(* Logix 5000 project; controller ProyectoIntegrador Emulate 5570 rev 30.11; software revision 30.00 *)

TASK MainTask (continuous, watchdog 500 ms) : MainProgram

MODULES
   Local : Emulate 5570 (ICP 2, rev 30.11)
      IO_module : vendor 1 type 0 code 15 (ICP 3, rev 1.1, Output RPI 150 ms)
END_MODULES

PROGRAM MainProgram   (* main routine MainRoutine *)
VAR
   Action_000 : SFC_ACTION := (Status := 16#0020_0000, PauseTimer := 1);
   Action_001 : SFC_ACTION := (Status := 16#0020_0000, PauseTimer := 1);
   Action_002 : SFC_ACTION := (Status := 16#0020_0000, PauseTimer := 1);
   Action_003 : SFC_ACTION := (Status := 16#0020_0000, PauseTimer := 1);
   Action_004 : SFC_ACTION := (Status := 16#0020_0000, PauseTimer := 1);
   Action_005 : SFC_ACTION := (Status := 16#0020_0000, PauseTimer := 1);
   Action_006 : SFC_ACTION := (Status := 16#0020_0000, PauseTimer := 1);
   Action_007 : SFC_ACTION := (Status := 16#0020_0000, PauseTimer := 1);
   Action_008 : SFC_ACTION := (Status := 16#0020_0000, PauseTimer := 1);
   Action_009 : SFC_ACTION := (Status := 16#0020_0000, PauseTimer := 1);
   Action_010 : SFC_ACTION := (Status := 16#0020_0000, PauseTimer := 1);
   Action_011 : SFC_ACTION := (Status := 16#0020_0000, PauseTimer := 1);
   Action_012 : SFC_ACTION := (Status := 16#0020_0000, PauseTimer := 1);
   Action_013 : SFC_ACTION := (Status := 16#0020_0000, PauseTimer := 1);
   Action_014 : SFC_ACTION := (Status := 16#0020_0000, PauseTimer := 1);
   C1b : BOOL;   // Moves Cilinder 1 backward
   C1f : BOOL;   // Move cilinder 1 forward
   C2b : DINT;   // Move the cilinder 2 backwards
   C2f : BOOL;   // Move the cilinder 2 forward
   Clasif : BOOL;   // Encender/Apagar Classificador
   Compressor : BOOL;   // Encender/Apagar Compressor
   Lavdo : BOOL;   // Encender/Apagar Lavado
   lConv : BOOL;   // Sensor de cajas conveyor belt 3 (vegetal grande)
   lCount : DINT;   // Large box counter
   mConv : BOOL;
   mCount : DINT;   // Medium Boxes count
   RC5 : BOOL;   // Encender/Apagar roller conveyor 4
   RC_1 : BOOL;   // Encender/Apagar roller conveyor 1
   RC_2 : BOOL;   // Encender/Apagar roller conveyor 2
   RC_3 : BOOL;   // Encender/Apagar roller conveyor 3
   RC_4 : BOOL;   // Encender/Apagar roller conveyor 4
   S1_C1 : BOOL;   // Cilindro 1 recogido
   S1_C2 : BOOL;   // Sensor 1 final de carrera cilindro2
   S2_C1 : BOOL;   // Sensor 2 final de carrera cilindro 1
   S2_C2 : BOOL;   // Sensor 2 final de carrera cilindro 2
   S_clasif : DINT;   // Sensor para clasificacion de empaque
   sConv : BOOL;
   sCount : DINT;   // Small Boxes Count
   Secado : BOOL;   // Encender/Apagar Secado
   Start : BOOL;   // Inicio del proceso
   Step_000 : SFC_STEP := (Status := 16#0020_0000, PauseTimer := 1);
   Step_001 : SFC_STEP := (Status := 16#0020_0000, PauseTimer := 1);
   Step_002 : SFC_STEP := (Status := 16#0020_0000, PauseTimer := 1);
   Step_003 : SFC_STEP := (Status := 16#0020_0000, PauseTimer := 1);
   Step_004 : SFC_STEP := (Status := 16#0020_0000, PauseTimer := 1);
   Step_005 : SFC_STEP := (Status := 16#0020_0000, PauseTimer := 1);
   Step_006 : SFC_STEP := (Status := 16#0020_0000, PauseTimer := 1);
   Step_007 : SFC_STEP := (Status := 16#0020_0000, PauseTimer := 1);
   Step_008 : SFC_STEP := (Status := 16#0020_0000, PauseTimer := 1);
   Step_009 : SFC_STEP := (Status := 16#0020_0000, PauseTimer := 1);
   Step_010 : SFC_STEP := (Status := 16#0020_0000, PauseTimer := 1);
   Step_011 : SFC_STEP := (Status := 16#0020_0000, PauseTimer := 1);
   Step_012 : SFC_STEP := (Status := 16#0020_0000, PauseTimer := 1);
   Step_013 : SFC_STEP := (Status := 16#0020_0000, PauseTimer := 1);
   Step_014 : SFC_STEP := (Status := 16#0020_0000, PauseTimer := 1);
   Step_015 : SFC_STEP := (Status := 16#0020_0000, PauseTimer := 1);
   Step_016 : SFC_STEP := (Status := 16#0020_0000, PauseTimer := 1);
   Step_017 : SFC_STEP := (Status := 16#0020_0000, PauseTimer := 1);
   Step_018 : SFC_STEP := (Status := 16#0020_0000, PauseTimer := 1);
   Step_021 : SFC_STEP := (Status := 16#0020_0000, PauseTimer := 1);
   Step_022 : SFC_STEP := (Status := 16#0020_0000, PauseTimer := 1);
   Step_023 : SFC_STEP := (Status := 16#0020_0000, PauseTimer := 1);
   Step_024 : SFC_STEP := (Status := 16#0020_0000, PauseTimer := 1);
   Step_025 : SFC_STEP := (Status := 16#0020_0000, PauseTimer := 1);
   Step_031 : SFC_STEP := (Status := 16#0020_0000, PauseTimer := 1);
   Step_041 : SFC_STEP := (Status := 16#0020_0000, PauseTimer := 1);
   Step_042 : SFC_STEP := (Status := 16#0020_0000, PauseTimer := 1);
   Step_100 : SFC_STEP := (Status := 16#0020_0000, PauseTimer := 1);
   Step_101 : SFC_STEP := (Status := 16#0020_0000, PauseTimer := 1);
   Step_102 : SFC_STEP := (Status := 16#0020_0000, PauseTimer := 1);
   Step_103 : SFC_STEP := (Status := 16#0020_0000, PauseTimer := 1);
   Stop : BOOL;   // Stop Button
   Tran_000 : BOOL;
   Tran_001 : BOOL;
   Tran_002 : BOOL;
   Tran_003 : BOOL;
   Tran_004 : BOOL;
   Tran_005 : BOOL;
   Tran_006 : BOOL;
   Tran_007 : BOOL;
   Tran_008 : BOOL;
   Tran_009 : BOOL;
   Tran_010 : BOOL;
   Tran_011 : BOOL;
   Tran_012 : BOOL;
   Tran_016 : BOOL;
   Tran_017 : BOOL;
   Tran_018 : BOOL;
   Tran_019 : BOOL;
   Volcar : BOOL;   // Encendr/Apagar volcador
END_VAR

ROUTINE Distribution   (* sequential function chart *)
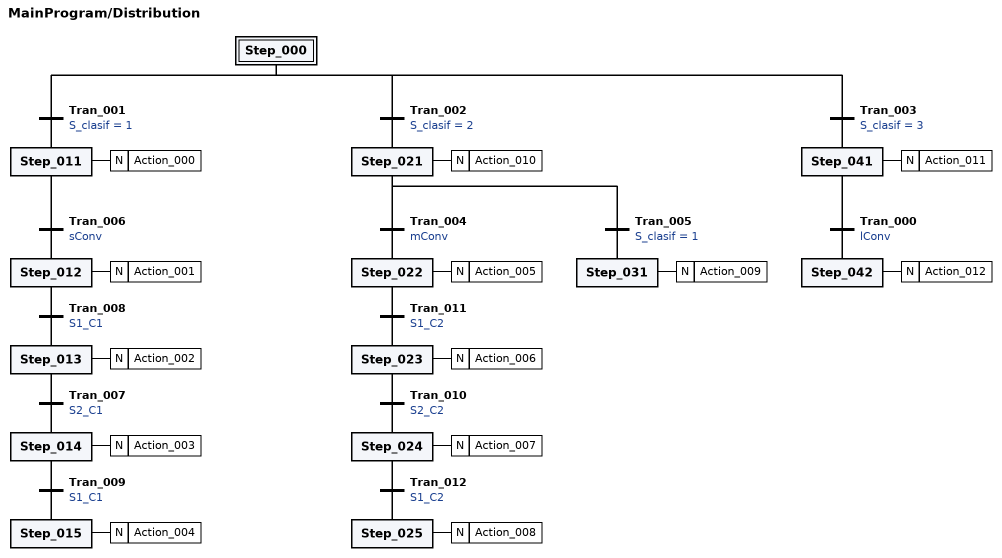
   // If the boxes
   // are medium
   // If the boxes
   // are small
   // If the boxes
   // are large
   // Sink
   // Transition
   // Pneumatic
   // divider G7
   // Sink
   // Transition
   // Sink
   // Transition
   // Discuss
   // with group
   // !!!
   // Should we have BC1, BC2 and BC3 always
   // turned on ??
   INITIAL_STEP Step_000:
   END_STEP
   TRANSITION Tran_001 FROM Step_000 TO Step_011
      := S_clasif = 1
         
   END_TRANSITION
   TRANSITION Tran_002 FROM Step_000 TO Step_021
      := S_clasif = 2
         
   END_TRANSITION
   TRANSITION Tran_003 FROM Step_000 TO Step_041
      := S_clasif = 3
         
   END_TRANSITION
   STEP Step_011:
      ACTION Action_000 (N):
         (* Move the rolling
         conveyor 5 forward*)
         RC5 := 1;
      END_ACTION
   END_STEP
   STEP Step_021:
      ACTION Action_010 (N):
         (* Move the rolling
         conveyor 5 forward*)
         RC5 := 1;
      END_ACTION
   END_STEP
   TRANSITION Tran_006 FROM Step_011 TO Step_012
      := sConv
   END_TRANSITION
   STEP Step_041:
      ACTION Action_011 (N):
         (* Move the rolling
         conveyor 5 forward*)
         RC5 := 1;
      END_ACTION
   END_STEP
   STEP Step_012:
      ACTION Action_001 (N):
         RC5 := 0;
         (*If the cilinder isnt
         in its back position
         move it there *)
         IF not S1_C1 THEN
             C1b := 1;
         END_IF;
         
      END_ACTION
   END_STEP
   TRANSITION Tran_004 FROM Step_021 TO Step_022
      := mConv
   END_TRANSITION
   TRANSITION Tran_005 FROM Step_021 TO Step_031
      := S_clasif = 1
         
   END_TRANSITION
   TRANSITION Tran_000 FROM Step_041 TO Step_042
      := lConv
   END_TRANSITION
   TRANSITION Tran_008 FROM Step_012 TO Step_013
      := S1_C1
         
   END_TRANSITION
   STEP Step_022:
      ACTION Action_005 (N):
         RC5 := 0;
         (*If the cilinder isnt
         in its back position
         move it there *)
         IF not S1_C2  THEN
             C2b := 1;
         END_IF;
         
      END_ACTION
   END_STEP
   STEP Step_031:
      ACTION Action_009 (N):
         (* We have a small box while we are
         moving a medium, so wait for 1 box
         to pass and then activate
         Step 004 *)
      END_ACTION
   END_STEP
   STEP Step_042:
      ACTION Action_012 (N):
         RC5 := 0;
         //Ativate start action and
         // BC3 action X_100 := 1 ;
         //Update the count
         lCount := lCount + 1 ;
      END_ACTION
   END_STEP
   STEP Step_013:
      ACTION Action_002 (N):
         // Turn off cilinder 1 back
         C1b := 0;
         // Turn on cilinder 1 forward
         C1f := 1;
      END_ACTION
   END_STEP
   TRANSITION Tran_011 FROM Step_022 TO Step_023
      := S1_C2
         
   END_TRANSITION
   TRANSITION Tran_007 FROM Step_013 TO Step_014
      := S2_C1
         
   END_TRANSITION
   STEP Step_014:
      ACTION Action_003 (N):
         //Turn off cilinder 1 forward
         C1f:=0;
         // Turn on cilinder 1 back
         C1b:=1;
      END_ACTION
   END_STEP
   STEP Step_023:
      ACTION Action_006 (N):
         // Turn off cilinder 2 back
         C2b := 0;
         // Turn on cilinder 2 forward
         C2f := 1;
      END_ACTION
   END_STEP
   TRANSITION Tran_009 FROM Step_014 TO Step_015
      := S1_C1
   END_TRANSITION
   TRANSITION Tran_010 FROM Step_023 TO Step_024
      := S2_C2
         
         
   END_TRANSITION
   STEP Step_015:
      ACTION Action_004 (N):
         //Turn off cilinder 1 back
         C1b:=0;
         //Ativate start action and
         // BC1 action X_100 := 1 ;
         //Update the count
         sCount := sCount + 1 ;
      END_ACTION
   END_STEP
   STEP Step_024:
      ACTION Action_007 (N):
         //Turn off cilinder 2 forward
         C2f:=0;
         // Turn on cilinder 2 back
         C2b:=1;
      END_ACTION
   END_STEP
   TRANSITION Tran_012 FROM Step_024 TO Step_025
      := S1_C2
   END_TRANSITION
   STEP Step_025:
      ACTION Action_008 (N):
         //Turn off cilinder 1 back
         C1b:=0;
         //Ativate start action and
         // BC2 action X_100 := 1 ;
         //Update the count
         mCount := mCount + 1 ;
         
         //What if we push more than 1 box ??
         // Go back to counting sensors ?
      END_ACTION
   END_STEP
END_ROUTINE

ROUTINE Main   (* sequential function chart *)
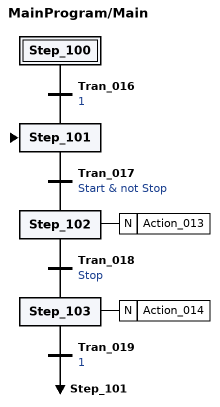
   // Look how to enable and disable
   // G7, might have to change
   // Classfier G7 to a macro ?
   // Change to
   // Rising Edge
   // - Look up
   // Guide
   // Change to
   // Rising Edge
   // - Look up
   // Guide
   // And with negative might help
   // but not perfect
   // Do we turn on all of these
   // while the button is pressed or
   // should we otimize in some
   // way ?
   INITIAL_STEP Step_100:
   END_STEP
   TRANSITION Tran_016 FROM Step_100 TO Step_101
      := 1
   END_TRANSITION
   STEP Step_101:
   END_STEP
   TRANSITION Tran_017 FROM Step_101 TO Step_102
      := Start & not Stop
   END_TRANSITION
   STEP Step_102:
      ACTION Action_013 (N):
         Volcar := 1;
         RC_1 := 1;
         RC_2 := 1;
         RC_3 := 1;
         RC_4 := 1;
         Lavdo := 1;
         Secado := 1;
         Clasif := 1;
         Compressor := 1;
         (*Activate Classifier G7*)
      END_ACTION
   END_STEP
   TRANSITION Tran_018 FROM Step_102 TO Step_103
      := Stop
   END_TRANSITION
   STEP Step_103:
      ACTION Action_014 (N):
         Volcar := 0;
         RC_1 := 0;
         RC_2 := 0;
         RC_3 := 0;
         RC_4 := 0;
         Lavdo := 0;
         Secado := 0;
         Clasif := 0;
         Compressor := 0;
         (*Deactivate Classifier G7*)
      END_ACTION
   END_STEP
   TRANSITION Tran_019 FROM Step_103 TO Step_101
      := 1
   END_TRANSITION
END_ROUTINE

ROUTINE MainRoutine   (* ladder *)
END_ROUTINE
END_PROGRAM
